// TIA Portal project "VascheFB" (V16)

(* hardware
DEVICE "S7-1200 station_1"  S7-1200 Station
   slot 0: "Telaio di montaggio_0"  S7-1200 Rack  Rack  V1.0
   slot 1: "PLC_1"  CPU 1214C DC/DC/DC  6ES7 214-1AG40-0XB0  V4.1
*)

// ===== PLC "PLC_1"  CPU 1214C DC/DC/DC =====

VAR_GLOBAL   // PLC tag table "Tabella delle variabili standard"
   "START" AT %I0.0 : Bool;
   "L1" AT %I0.1 : Bool;
   "L2" AT %I0.2 : Bool;
   "L3" AT %I0.3 : Bool;
   "P1" AT %Q0.1 : Bool;
   "P2" AT %Q0.2 : Bool;
END_VAR

VAR_GLOBAL CONSTANT   // PLC tag table "Tabella delle variabili standard"
   "TEMPO_TRASCORSO_ON_1" : Time := T#5s;
   "TEMPO_TRASCORSO_ON_Delta_1" : Time := T#10s;
   "TEMPO_TRASCORSO_ON_2" : Time := T#30s;
   "TEMPO_TRASCORSO_ON_Delta_2" : Time := T#15s;
   "TEMPO_TRASCORSO_Pausa" : Time := T#30s;
END_VAR

DATA_BLOCK "Vasche_DB"   // DB1
{ S7_Optimized_Access := 'TRUE' }
VERSION : 0.1
// stored: InstanceOfName Vasche
"Vasche"
BEGIN
END_DATA_BLOCK

FUNCTION_BLOCK "Vasche"   // FB1, LAD
{ S7_Optimized_Access := 'TRUE' }
VERSION : 0.1
   VAR_INPUT
      START : Bool;
      L1 : Bool;
      L2 : Bool;
      L3 : Bool;
      TEMPO_TRASCORSO_ON_1 : Time;
      TEMPO_TRASCORSO_ON_Delta_1 : Time;
      TEMPO_TRASCORSO_ON_2 : Time;
      TEMPO_TRASCORSO_ON_Delta_2 : Time;
      TEMPO_Trascorso_Pausa : Time;
   END_VAR
   VAR_OUTPUT
      P1 : Bool;
      P2 : Bool;
   END_VAR
   VAR RETAIN
      HOME : Bool := true;
      POMPE_ON_1 : Bool;
      POMPA_2_OFF_n1 : Bool;
      POMPE_OFF : Bool;
      POMPE_ON_2 : Bool;
      POMPA_2_OFF_n2 : Bool;
   END_VAR
   VAR
      IEC_Timer_0_Instance_1 : TON_TIME;
      IEC_Timer_0_Instance_2 : TON_TIME;
      IEC_Timer_0_Instance_3 : TON_TIME;
      IEC_Timer_0_Instance_4 : TON_TIME;
      IEC_Timer_0_Instance_5 : TON_TIME;
   END_VAR
BEGIN

REGION Network 1
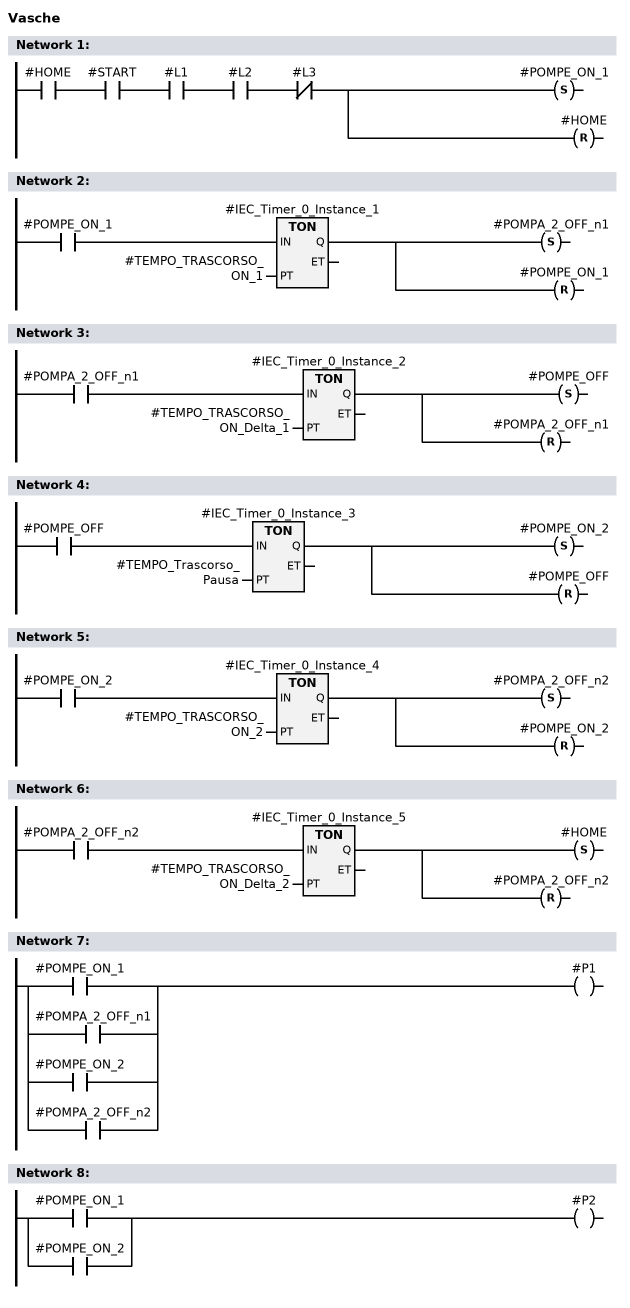
   RUNG wire#powerrail
      Contact( #HOME )
      Contact( #START )
      Contact( #L1 )
      Contact( #L2 )
      I_Contact( #L3 )
      wire#w1
      S_Coil( #POMPE_ON_1 )
   END_RUNG
   RUNG wire#w1
      R_Coil( #HOME )
   END_RUNG
   // the same network as SCL:
   IF #HOME AND #START AND #L1 AND #L2 AND NOT #L3 THEN
       #POMPE_ON_1 := TRUE;
       #HOME := FALSE;
   END_IF;
END_REGION

REGION Network 2
   #IEC_Timer_0_Instance_1(IN := #POMPE_ON_1, PT := #TEMPO_TRASCORSO_ON_1);   // TON
   IF #IEC_Timer_0_Instance_1.Q THEN
       #POMPA_2_OFF_n1 := TRUE;
       #POMPE_ON_1 := FALSE;
   END_IF;
END_REGION

REGION Network 3
   #IEC_Timer_0_Instance_2(IN := #POMPA_2_OFF_n1, PT := #TEMPO_TRASCORSO_ON_Delta_1);   // TON
   IF #IEC_Timer_0_Instance_2.Q THEN
       #POMPE_OFF := TRUE;
       #POMPA_2_OFF_n1 := FALSE;
   END_IF;
END_REGION

REGION Network 4
   #IEC_Timer_0_Instance_3(IN := #POMPE_OFF, PT := #TEMPO_Trascorso_Pausa);   // TON
   IF #IEC_Timer_0_Instance_3.Q THEN
       #POMPE_ON_2 := TRUE;
       #POMPE_OFF := FALSE;
   END_IF;
END_REGION

REGION Network 5
   #IEC_Timer_0_Instance_4(IN := #POMPE_ON_2, PT := #TEMPO_TRASCORSO_ON_2);   // TON
   IF #IEC_Timer_0_Instance_4.Q THEN
       #POMPA_2_OFF_n2 := TRUE;
       #POMPE_ON_2 := FALSE;
   END_IF;
END_REGION

REGION Network 6
   #IEC_Timer_0_Instance_5(IN := #POMPA_2_OFF_n2, PT := #TEMPO_TRASCORSO_ON_Delta_2);   // TON
   IF #IEC_Timer_0_Instance_5.Q THEN
       #HOME := TRUE;
       #POMPA_2_OFF_n2 := FALSE;
   END_IF;
END_REGION

REGION Network 7
   RUNG wire#powerrail
      Contact( #POMPE_ON_1 )
      wire#w1
      Coil( #P1 )
   END_RUNG
   RUNG wire#powerrail
      Contact( #POMPA_2_OFF_n1 )
   END_RUNG wire#w1
   RUNG wire#powerrail
      Contact( #POMPE_ON_2 )
   END_RUNG wire#w1
   RUNG wire#powerrail
      Contact( #POMPA_2_OFF_n2 )
   END_RUNG wire#w1
   // the same network as SCL:
   #P1 := #POMPE_ON_1 OR #POMPA_2_OFF_n1 OR #POMPE_ON_2 OR #POMPA_2_OFF_n2;
END_REGION

REGION Network 8
   RUNG wire#powerrail
      Contact( #POMPE_ON_1 )
      wire#w1
      Coil( #P2 )
   END_RUNG
   RUNG wire#powerrail
      Contact( #POMPE_ON_2 )
   END_RUNG wire#w1
   // the same network as SCL:
   #P2 := #POMPE_ON_1 OR #POMPE_ON_2;
END_REGION
END_FUNCTION_BLOCK

ORGANIZATION_BLOCK "Main"   // OB1, LAD, ProgramCycle
TITLE = "Main Program Sweep (Cycle)"
{ S7_Optimized_Access := 'TRUE' }
VERSION : 0.1
   VAR_INPUT
      Initial_Call : Bool;   // Initial call of this OB
      Remanence : Bool;   // =True, if remanent data are available
   END_VAR
BEGIN

REGION Network 1
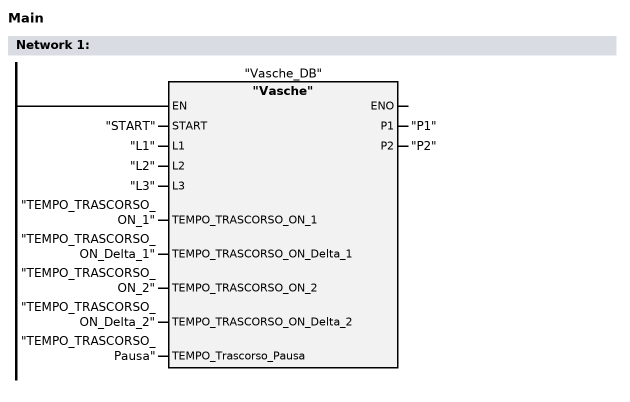
   RUNG wire#powerrail
      "Vasche_DB"(START := "START", L1 := "L1", L2 := "L2", L3 := "L3", TEMPO_TRASCORSO_ON_1 := "TEMPO_TRASCORSO_ON_1", TEMPO_TRASCORSO_ON_Delta_1 := "TEMPO_TRASCORSO_ON_Delta_1", TEMPO_TRASCORSO_ON_2 := "TEMPO_TRASCORSO_ON_2", TEMPO_TRASCORSO_ON_Delta_2 := "TEMPO_TRASCORSO_ON_Delta_2", TEMPO_Trascorso_Pausa := "TEMPO_TRASCORSO_Pausa", P1 => "P1", P2 => "P2")
   END_RUNG
   // the same network as SCL:
   "Vasche_DB"(START := "START",   // "Vasche"
               L1 := "L1",
               L2 := "L2",
               L3 := "L3",
               TEMPO_TRASCORSO_ON_1 := "TEMPO_TRASCORSO_ON_1",
               TEMPO_TRASCORSO_ON_Delta_1 := "TEMPO_TRASCORSO_ON_Delta_1",
               TEMPO_TRASCORSO_ON_2 := "TEMPO_TRASCORSO_ON_2",
               TEMPO_TRASCORSO_ON_Delta_2 := "TEMPO_TRASCORSO_ON_Delta_2",
               TEMPO_Trascorso_Pausa := "TEMPO_TRASCORSO_Pausa",
               P1 => "P1",
               P2 => "P2");
END_REGION
END_ORGANIZATION_BLOCK